Fanuc TP program (LS listing): KPPREP.LS

/PROG  KPPREP
/ATTR
OWNER		= MNEDITOR;
COMMENT		= "KAREL pose probe prep";
PROG_SIZE	= 0;
CREATE		= DATE 26-01-01  TIME 00:00:00;
MODIFIED	= DATE 26-01-01  TIME 00:00:00;
FILE_NAME	= ;
VERSION		= 0;
LINE_COUNT	= 13;
MEMORY_SIZE	= 0;
PROTECT		= READ_WRITE;
TCD:  STACK_SIZE	= 0,
      TASK_PRIORITY	= 50,
      TIME_SLICE	= 0,
      BUSY_LAMP_OFF	= 0,
      ABORT_REQUEST	= 0,
      PAUSE_REQUEST	= 0;
DEFAULT_GROUP	= 1,*,*,*,*;
CONTROL_CODE	= 00000000 00000000;
/MN
   1:  UFRAME_NUM=0 ;
   2:  UTOOL_NUM=1 ;
   3:  PR[96]=LPOS    ;
   4:  PR[91]=LPOS    ;
   5:  PR[90]=LPOS    ;
   6:  PR[92]=LPOS    ;
   7:  PR[95]=LPOS    ;
   8:  PR[93]=LPOS    ;
   9:  PR[89]=LPOS    ;
  10:  PR[99]=LPOS    ;
  11:  PR[98]=LPOS    ;
  12:  PR[97]=LPOS    ;
  13:  PR[94]=LPOS    ;
/POS
/END
